Staubli VAL3: CanProduct.pgx

public program CanProduct(num& x_nWorkPlace (dimensions=1))
begin
  //等待IO响应



  //第一工位
  if dDio["In1_bPrdSta1"]==true
    delay(0.2)
    if watch(dDio["In1_bPrdSta1"]==true,0.1)
      if watch(dDio["In1_bPrdSta1"]==false,2)
        logMsg("In1_bPrdSta1触发:工位1信号被触发")
        //      x_bCanProuct[1]=true
        x_nWorkPlace=1
        return
      endIf
    endIf
  endIf

  //第二工位
  if dDio["In1_bPrdSta2"]==true
    delay(0.2)
    if watch(dDio["In1_bPrdSta2"]==true,0.1)
      if watch(dDio["In1_bPrdSta2"]==false,2)
        logMsg("In1_bPrdSta2触发:工位2信号被触发")
        //x_bCanProuct[2]=true
        x_nWorkPlace=2
        return
      endIf
    endIf
  endIf


  //第三工位
  if dDio["In2_bPrdSta3"]==true
    delay(0.2)
    if watch(dDio["In2_bPrdSta3"]==true,0.1)
      if watch(dDio["In2_bPrdSta3"]==false,2)
        logMsg("In2_bPrdSta3触发:工位3信号被触发")
        //      x_bCanProuct[3]=true
        x_nWorkPlace=3
        return
      endIf
    endIf
  endIf

  //第四工位
  if dDio["In2_bPrdSta4"]==true
    delay(0.2)
    if watch(dDio["In2_bPrdSta4"]==true,0.1)
      //      x_bCanProuct[4]=true
      if watch(dDio["In2_bPrdSta4"]==false,2)
        logMsg("In2_bPrdSta4触发:工位4信号被触发")
        x_nWorkPlace=4
        return
      endIf
    endIf
  endIf



end
